FUNCTION CB_real_to_word : word


TITLE = ' Convert a real into a word '
VERSION : '1.0'
AUTHOR  : CB
NAME    : realWord
FAMILY  : TNI

VAR_INPUT
    IN : REAL;
END_VAR

VAR_TEMP

END_VAR

BEGIN

CB_real_to_word := INT_TO_WORD(REAL_TO_INT(IN));

END_FUNCTION
